PROGRAM MAIN
VAR
	fbBanner			: FB_BannerK50;
	
	Toggle				: BOOL := FALSE;
END_VAR

fbBanner();

END_PROGRAM

(* stored: Version 1.1.0.1, ProductVersion 3.1.4024.11
   POU MAIN: Id {1f5d730c-9e96-4a11-b15c-ef2848a86c90}, SpecialFunc None *)
